TYPE ST_ProBoxSafetyVerticalConv :
STRUCT
	Inputs	AT %I* : ST_ProBoxSafetyInputsVerticalConv;
	Outputs AT %Q* : ST_ProBoxSafetyOutputsVerticalConv;
END_STRUCT
END_TYPE

(* stored: Version 1.1.0.1, ProductVersion 3.1.4024.4
   DUT ST_ProBoxSafetyVerticalConv: Id {891d9bf9-e09f-4c3e-9833-d1f3498f111b} *)
